// TwinCAT 3 PLC project Listener
// ProgramVersion: 3.1.4021.2
// libraries:
//   Tc2_Standard, * (Beckhoff Automation GmbH)
//   Tc2_System, * (Beckhoff Automation GmbH)
//   Tc2_TcpIp, * (Beckhoff Automation GmbH)
//   Tc2_Utilities, * (Beckhoff Automation GmbH)
//   Tc3_EventLogger, * (Beckhoff Automation GmbH)
//   Tc3_JsonXml, * (Beckhoff Automation GmbH)
//   Tc3_Module, * (Beckhoff Automation GmbH)
// project tree:
//   DUTs/ ST_EventInfo.TcDUT, E_LogEventType.TcDUT (not stored), ST_PendingEvent.TcDUT (not stored)
//   GVLs/ GVL_Logger.TcGVL
//   / ListenerTask.TcTTO
//   POUs/ FB_LogHandler.TcPOU, F_ConvertTicksToUnixTimestamp.TcPOU (not stored), F_SendUDPMessage.TcPOU (not stored), MAIN.TcPOU, FB_Listener.TcPOU
// (motion and I/O tree: see PLC project publisher)
// real-time tasks:
//   TASK PublisherTask: cycle T#10ms, priority 20, ADS port 350
//   TASK ListenerTask: cycle T#10ms, priority 1, ADS port 351

CONFIGURATION Listener
    RESOURCE PLC ON TwinCAT3
        TASK ListenerTask(INTERVAL := T#10ms, PRIORITY := 1);
        PROGRAM MAIN WITH ListenerTask : MAIN;
    END_RESOURCE
END_CONFIGURATION

// ---- DUTs/ST_EventInfo.TcDUT
TYPE ST_EventInfo :
STRUCT
	(* 
		Message or Alarm{Cleared,Confirmed,Raised} event information
		
		Note that elements here do not follow the usual Hungarian notation / 
		variable-type-prefixing naming convention due to the member names being
		used directly in the generation of the JSON document.
	*)
	
	{attribute 'pytmc' := '
		pv: Schema
		io: i
		field: DESC Schema string
	'}
	schema		:	STRING := 'twincat-event-0';
	  
	{attribute 'pytmc' := '
		pv: Timestamp 
		io: i
		field: DESC Unix timestamp
	'}
  	ts			:	LREAL;
  
	{attribute 'pytmc' := '
		pv: Severity
		io: i
		field: DESC TcEventSeverity	
		field: ZRST Verbose
		field: ONST Info
		field: TWST Warning
		field: THST Error
	'}
	severity	:	TcEventSeverity;
	
	{attribute 'pytmc' := '
		pv: MessageID
		io: i
		field: DESC TwinCAT Message ID	
	'}
	id			:	UDINT;

	{attribute 'pytmc' := '
		pv: EventClass
		io: i
		field: DESC TwinCAT Event class	
	'}
	event_class		:	STRING;
		
	{attribute 'pytmc' := '
		pv: Message
		io: i
	'}
	msg			:	 T_MaxString;

	{attribute 'pytmc' := '
		pv: Source
		io: i
	'}
	source		:	 T_MaxString;
	
	{attribute 'pytmc' := '
		pv: EventType
		io: i
		field: DESC The event type
	'}
	event_type	:	 E_LogEventType;
	
	{attribute 'pytmc' := '
		pv: MessageJSON
		io: i
		field: DESC Metadata with the message	
	'}
	json 		:	STRING(10000);
	(* 
	NOTE: this JSON gets inserted as an escaped string in the "json" key.
	TODO: it may be possible to use `fbJson.AddRawObject`, but this would
		  require us to switch back to creating the JSON in a more manual
		  way with AddKey/AddInt (and such).
	*)		 

END_STRUCT
END_TYPE

// ---- GVLs/GVL_Logger.TcGVL
VAR_GLOBAL
	cLogHost		:	T_IPv4Addr	:= '172.21.148.141';
	iLogPort		:	UINT		:= 50000;
	sPlcHostname	:	STRING		:= 'unknown';
	
	(* Ref: https://infosys.beckhoff.com/english.php?content=../content/1033/tcpipserver/html/TcPlcLibTcpIp_FB_SocketUdpSendTo.htm
		TODO: Activate the "Replace constants" option in the
		TwinCAT PLC Control->"Project->Options...->Build" dialog window. 
	*)
	TCPADS_MAXUDP_BUFFSIZE : UDINT :=10000;
	
END_VAR

// ---- POUs/MAIN.TcPOU
PROGRAM MAIN
VAR
	{attribute 'pytmc' := '
		pv: Logging
	'}
	fbLogHandler : FB_LogHandler;
END_VAR

fbLogHandler();

END_PROGRAM

// ---- POUs/FB_LogHandler.TcPOU
FUNCTION_BLOCK FB_LogHandler
VAR_INPUT
END_VAR
VAR_OUTPUT
END_VAR

VAR
	
	bInitialized	:	BOOL	:= FALSE;
	fbGetHostName	:	FB_GetHostName := (bExecute := TRUE, sNetID := ''); //Acquires name of the PLC
	bHostnameSet	:	BOOL	:= FALSE;

	{attribute 'pytmc' := '
		pv: ADS
	'}
	fbTcAdsListener : FB_Listener;	
	
	{attribute 'pytmc' := '
		pv: Router
	'}
	fbTcRouterListener : FB_Listener;	
	
	{attribute 'pytmc' := '
		pv: RTime
	'}
	fbTcRTimeListener : FB_Listener;	
	
	{attribute 'pytmc' := '
		pv: System
	'}
	fbTcSystemListener : FB_Listener;
	
	{attribute 'pytmc' := '
		pv: Windows
	'}
	fbWindowsListener : FB_Listener;	

	{attribute 'pytmc' := '
		pv: LCLS
	'}
	fbLCLSListener 	: FB_Listener;	

	fbListener		:	REFERENCE TO FB_Listener;
	fbListeners		: 	ARRAY [0..nNumListeners - 1] OF POINTER TO FB_Listener;
	
	// Default minimum severity for subscriptions
	eMinSeverity	:	TcEventSeverity := TcEventSeverity.Verbose;	
	
	{attribute 'naming' := 'omit'}
	rtReset				:	R_TRIG; //Reset trigger
	bReset				:	BOOL;
		
	fbSocket	   		:	FB_ConnectionlessSocket;
	
	nI: UINT;
END_VAR

VAR CONSTANT
	nNumListeners		:	UINT	:= 6;
END_VAR

IF NOT bInitialized THEN 
	bInitialized := TRUE;
	fbTcAdsListener.Configure(i_EventClass:=TC_EVENT_CLASSES.TcGeneralAdsEventClass, i_MinSeverity:=eMinSeverity, i_fbSocket:=ADR(fbSocket));
	fbTcRouterListener.Configure(i_EventClass:=TC_EVENT_CLASSES.TcRouterEventClass, i_MinSeverity:=eMinSeverity, i_fbSocket:=ADR(fbSocket));
	fbTcRTimeListener.Configure(i_EventClass:=TC_EVENT_CLASSES.TcRTimeEventClass, i_MinSeverity:=eMinSeverity, i_fbSocket:=ADR(fbSocket));
	fbTcSystemListener.Configure(i_EventClass:=TC_EVENT_CLASSES.TcSystemEventClass, i_MinSeverity:=eMinSeverity, i_fbSocket:=ADR(fbSocket));
	fbWindowsListener.Configure(i_EventClass:=TC_EVENT_CLASSES.Win32EventClass, i_MinSeverity:=eMinSeverity, i_fbSocket:=ADR(fbSocket));
	fbLCLSListener.Configure(i_EventClass:=TC_EVENT_CLASSES.LCLSLoggingEvent, i_MinSeverity:=eMinSeverity, i_fbSocket:=ADR(fbSocket));

	fbListeners[0] := ADR(fbTcAdsListener);
	fbListeners[1] := ADR(fbTcRouterListener);
	fbListeners[2] := ADR(fbTcRTimeListener);
	fbListeners[3] := ADR(fbTcSystemListener);
	fbListeners[4] := ADR(fbWindowsListener);
	fbListeners[5] := ADR(fbLCLSListener);
END_IF 
	
IF NOT bHostnameSet THEN
	fbGetHostName();
	IF NOT (fbGetHostName.bBusy OR fbGetHostName.bError) THEN
		GVL_Logger.sPlcHostname := fbGetHostName.sHostName;
		bHostnameSet 			:= TRUE;
	END_IF
END_IF

(* Ensure the socket is ready for when JSON documents are emitted *)
rtReset(CLK:=bReset);

IF (rtReset.Q AND fbSocket.bEnable) OR fbSocket.bError THEN
	fbSocket(bEnable:=FALSE);
END_IF

fbSocket(
	nLocalPort:=0,
	bEnable:=TRUE,
	nMode:=CONNECT_MODE_ENABLEDBG,
);

(* Poke all of the listeners *)
FOR nI := 0 TO nNumListeners - 1 DO
	fbListener REF= fbListeners[nI]^;
	fbListener.Execute();
	fbListener.PublishEvents();
END_FOR

END_FUNCTION_BLOCK

// ---- POUs/FB_Listener.TcPOU
FUNCTION_BLOCK FB_Listener EXTENDS FB_ListenerBase
VAR_INPUT
END_VAR

VAR_OUTPUT
END_VAR

VAR
	nEventIdx			:	UINT := 0;
	nPendingEvents		:	UINT := 0;
	
	{attribute 'pytmc' := '
		pv: LogToVisualStudio
		io: io
	'}
	bLogToVisualStudio	:	BOOL := FALSE;
	
	{attribute 'pytmc' := '
		pv: MessagesSent
		io: i
	'}
	nCntMessagesSent 	: UDINT := 0;

	{attribute 'pytmc' := '
		pv: AlarmsRaised
		io: i
	'}
	nCntAlarmsRaised 	: UDINT := 0;
	
	{attribute 'pytmc' := '
		pv: AlarmsConfirmed
		io: i
	'}
	nCntAlarmsConfirmed : UDINT := 0;
	
	{attribute 'pytmc' := '
		pv: AlarmsCleared
		io: i
	'}
	nCntAlarmsCleared 	: UDINT := 0;
	
	{attribute 'pytmc' := '
		pv: MinSeverity
		io: io
	'}
	eMinSeverity	 	: TcEventSeverity;

	{attribute 'pytmc' := '
		pv: Log
	'}
	stEventInfo 		:	REFERENCE TO ST_EventInfo;

	stPendingEvents		:	ARRAY [0..nMaxEvents - 1] OF ST_PendingEvent;
	ipMessageConfig		:	ITcEventFilterConfig;
	fbSocket			:	POINTER TO FB_ConnectionlessSocket;
	bConfigured			:	BOOL	:= FALSE;
END_VAR

VAR_IN_OUT
	
END_VAR

VAR CONSTANT
	// The maximum number of events allowed *per-cycle*
	nMaxEvents			:	UINT := 10;
END_VAR

(*
	Configure an event class + severity
*)
METHOD Configure : HRESULT
VAR_INPUT
	i_EventClass 	:	GUID;
	i_MinSeverity	:	TcEventSeverity := TcEventSeverity.Verbose;
	i_fbSocket		:	POINTER TO FB_ConnectionlessSocket;	
END_VAR

VAR
	bSubscribed		:	BOOL := FALSE;
END_VAR
IF bSubscribed THEN
	Unsubscribe();
END_IF

THIS^.Subscribe(ADR(ipMessageConfig), 0);
bSubscribed 	:= TRUE;
eMinSeverity 	:= i_MinSeverity;
fbSocket	  	:= i_fbSocket;

IF (ipMessageConfig = 0) THEN
	Configure 	:= 1;
	bConfigured := FALSE;
ELSE
	ipMessageConfig.AddEventClass(i_EventClass, i_MinSeverity);
	Configure 	:= 0;
	bConfigured := TRUE;
END_IF
END_METHOD

METHOD OnAlarmCleared
VAR_INPUT
	fbEvent : REFERENCE TO FB_TcEvent;
END_VAR
(* Callback run from THIS^.Execute() *)
nCntAlarmsCleared := nCntAlarmsCleared + 1;
StoreEvent(fbEvent, eEventType:=E_LogEventType.AlarmCleared);
END_METHOD

METHOD OnAlarmConfirmed
VAR_INPUT
	fbEvent : REFERENCE TO FB_TcEvent;
END_VAR
(* Callback run from THIS^.Execute() *)
nCntAlarmsConfirmed := nCntAlarmsConfirmed + 1;
StoreEvent(fbEvent, eEventType:=E_LogEventType.AlarmConfirmed);
END_METHOD

METHOD OnAlarmRaised
VAR_INPUT
	fbEvent : REFERENCE TO FB_TcEvent;
END_VAR
(* Callback run from THIS^.Execute() *)
nCntAlarmsRaised := nCntAlarmsRaised + 1;
StoreEvent(fbEvent, eEventType:=E_LogEventType.AlarmRaised);
END_METHOD

METHOD OnMessageSent
VAR_INPUT
	fbEvent : REFERENCE TO FB_TcEvent;
END_VAR
(* Callback run from THIS^.Execute() *)
nCntMessagesSent := nCntMessagesSent + 1;
StoreEvent(fbEvent, eEventType:=E_LogEventType.MessageSent);
END_METHOD

METHOD PublishEvents : HRESULT
VAR
	fbJson				:	FB_JsonSaxWriter;
	fbJsonDataType		:	FB_JsonReadWriteDataType;
	sJsonDoc			:	STRING(10000);
	nEvent				:	UINT;
	stPendingEvent		:	REFERENCE TO ST_PendingEvent;
	stEventInfo			:	REFERENCE TO ST_EventInfo;
	fbRequestEventText	:	REFERENCE TO FB_RequestEventText;
END_VAR
IF nPendingEvents = 0 THEN
	RETURN;
END_IF

FOR nEvent := 0 TO nMaxEvents - 1 DO
	stPendingEvent REF= stPendingEvents[nEvent];
	IF NOT stPendingEvent.bInUse THEN
		CONTINUE;
	END_IF
	
	fbRequestEventText REF= stPendingEvent.fbRequestEventText;
	stEventInfo 	   REF= stPendingEvent.stEventInfo;
	
	IF fbRequestEventText.bError THEN 
		stEventInfo.Msg := '(Unable to retrieve message)';
	ELSIF NOT fbRequestEventText.bBusy THEN
		fbRequestEventText.GetString(stEventInfo.msg, SIZEOF(stEventInfo.msg));
	ELSE
		CONTINUE;
	END_IF
	
	IF bConfigured THEN
		// Generate the JSON message
		fbJson.ResetDocument();
		fbJsonDataType.AddJsonValueFromSymbol(fbJson, 'ST_EventInfo', SIZEOF(stEventInfo), ADR(stEventInfo));
		fbJson.CopyDocument(sJsonDoc, SIZEOF(sJsonDoc));
		
		//sJsonDoc := '{"message": "test"}';
		SendMessage(sMessage:=ADR(sJsonDoc));
	END_IF
	
	// Mark as not in use, and fill in this event in the next StoreEvent call
	nPendingEvents			:= nPendingEvents - 1;
	stPendingEvent.bInUse 	:= FALSE;
	nEventIdx 				:= nEvent;
	
END_FOR
END_METHOD

METHOD SendMessage : HRESULT
VAR_INPUT
	sMessage		:	POINTER TO STRING;
END_VAR

VAR
	sLogStr			:	T_MaxString;
END_VAR
(* For subclasses to override, if necessary *)
IF sMessage = 0 THEN
	RETURN;
END_IF

// Optionally log it to Visual Studio's message list
IF bLogToVisualStudio THEN
	 // Keep the message length under 255 (extended string function for LEFT/MID do not exist)
	STRNCPY(ADR(sLogStr), sMessage, MIN(220, SIZEOF(sLogStr)));
	ADSLOGSTR(
		msgCtrlMask := ADSLOG_MSGTYPE_HINT, 
		msgFmtStr   := '[Logger JSON Debug] %s', 
		strArg      := sLogStr
	); 
END_IF

IF fbSocket <> 0 THEN
	// And send it along to logstash
	F_SendUDPMessage(sMessage:=sMessage, fbSocket:=fbSocket^, 
					 sHost:=GVL_Logger.cLogHost, iPort:=GVL_Logger.iLogPort);
END_IF
END_METHOD

METHOD PRIVATE StoreEvent : HRESULT
VAR_INPUT
	fbEvent		:	REFERENCE TO FB_TcEvent;
	eEventType	:	E_LogEventType;
END_VAR

VAR
	stPendingEvent	:	REFERENCE TO ST_PendingEvent;
	stEventInfo		:	REFERENCE TO ST_EventInfo;
	nFailures		:	UINT := 0;
END_VAR
IF fbEvent.eSeverity < eMinSeverity THEN
	// Ignore all messages below the minimum severity
	RETURN;
ELSIF NOT __ISVALIDREF(fbEvent) THEN
	RETURN;
END_IF

// Find the next slot to use in stPendingEvents
WHILE stPendingEvents[nEventIdx].bInUse AND nFailures < nMaxEvents DO
	nFailures := nFailures + 1;
	IF ((nEventIdx := (nEventIdx + 1)) = nMaxEvents) THEN
		nEventIdx := 0;
	END_IF
END_WHILE

IF (nFailures = nMaxEvents) THEN
	ADSLOGSTR(
		msgCtrlMask := ADSLOG_MSGTYPE_ERROR, 
		msgFmtStr   := 'Logging message buffer full (%s)',
		strArg		:= UINT_TO_STRING(nMaxEvents),
	);
	RETURN;
END_IF

nPendingEvents			:=	nPendingEvents + 1;
nCntMessagesSent 		:=	nCntMessagesSent + 1;

stPendingEvent			REF= stPendingEvents[nEventIdx];
stEventInfo 			REF= stPendingEvent.stEventInfo;
stPendingEvent.bInUse 	:= TRUE;

stEventInfo.id 			:= fbEvent.nEventId;
stEventInfo.event_class	:= GUID_TO_STRING(fbEvent.EventClass);
stEventInfo.severity 	:= fbEvent.eSeverity;
stEventInfo.ts			:= F_ConvertTicksToUnixTimestamp(fbEvent.nTimestamp);
stEventInfo.source 		:= fbEvent.ipSourceInfo.sName;
stEventInfo.event_type	:= eEventType;

fbEvent.GetJsonAttribute(stEventInfo.json, SIZEOF(stEventInfo.json));
stPendingEvent.fbRequestEventText.Request(eventClass:=fbEvent.EventClass, nEventId:=fbEvent.nEventId, nLangId:=1033, ipArgs:=fbEvent.ipArguments);
END_METHOD

END_FUNCTION_BLOCK
